FUNCTION_BLOCK IORevPiDIO (* Digital I/O module for Revolution Pi by KUNBUS GmbH *)
  (* Standard: 61499-2; Description: Copyright (c) 2018 fortiss GmbH This program and the accompanying materials are made available under the terms of the Eclipse Public License 2.0 which is available at https://www.eclipse.org/legal/epl-2.0/ SPDX-License-Identifier: EPL-2.0 *)
  (* Version 1.0, 2018-04-22, Jos?? Cabral, fortiss GmbH *)
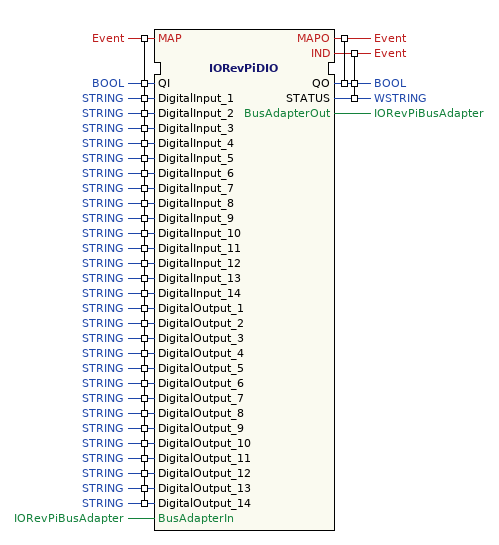
  EVENT_INPUT
    MAP WITH DigitalInput_1, DigitalInput_2, DigitalInput_5, DigitalInput_3, DigitalInput_4, DigitalInput_6, DigitalInput_7, DigitalInput_8, DigitalOutput_1, DigitalOutput_2, DigitalOutput_3, DigitalOutput_4, DigitalOutput_5, DigitalOutput_6, DigitalOutput_7, DigitalOutput_8, QI, DigitalInput_14, DigitalInput_13, DigitalInput_12, DigitalInput_11, DigitalInput_10, DigitalInput_9, DigitalOutput_9, DigitalOutput_10, DigitalOutput_11, DigitalOutput_12, DigitalOutput_13, DigitalOutput_14; (* Map Pins *)
  END_EVENT
  EVENT_OUTPUT
    MAPO WITH QO; (* Confirm Pin Mapping *)
    IND WITH QO, STATUS; (* Indication from Resource *)
  END_EVENT
  VAR_INPUT
    QI : BOOL; (* Event Input Qualifier *)
    DigitalInput_1 : STRING;
    DigitalInput_2 : STRING;
    DigitalInput_3 : STRING;
    DigitalInput_4 : STRING;
    DigitalInput_5 : STRING;
    DigitalInput_6 : STRING;
    DigitalInput_7 : STRING;
    DigitalInput_8 : STRING;
    DigitalInput_9 : STRING;
    DigitalInput_10 : STRING;
    DigitalInput_11 : STRING;
    DigitalInput_12 : STRING;
    DigitalInput_13 : STRING;
    DigitalInput_14 : STRING;
    DigitalOutput_1 : STRING;
    DigitalOutput_2 : STRING;
    DigitalOutput_3 : STRING;
    DigitalOutput_4 : STRING;
    DigitalOutput_5 : STRING;
    DigitalOutput_6 : STRING;
    DigitalOutput_7 : STRING;
    DigitalOutput_8 : STRING;
    DigitalOutput_9 : STRING;
    DigitalOutput_10 : STRING;
    DigitalOutput_11 : STRING;
    DigitalOutput_12 : STRING;
    DigitalOutput_13 : STRING;
    DigitalOutput_14 : STRING;
  END_VAR
  VAR_OUTPUT
    QO : BOOL; (* Event Output Qualifier *)
    STATUS : WSTRING; (* Service Status *)
  END_VAR
  SOCKETS
    BusAdapterIn : IORevPiBusAdapter;
  END_SOCKETS
  PLUGS
    BusAdapterOut : IORevPiBusAdapter;
  END_PLUGS
END_FUNCTION_BLOCK
